PROGRAM MAIN

END_PROGRAM

(* stored: Version 1.1.0.1, ProductVersion 3.1.4024.9
   POU MAIN: Id {55e5d4d9-4607-4a4e-b397-63e624f66e96}, SpecialFunc None *)
